# B&R Automation Studio project Parker_BMM_ST_V5_3147_V12 (part 28)

#### extruder.c - Implementation code
```c
/********************************************************************
 * COPYRIGHT --
 ********************************************************************
 * Program: extruder
 * File: extruder.c
 * Author: lij
 * Created: January 05, 2015
 ********************************************************************
 * Implementation of program extruder
 ********************************************************************/

#include <bur/plctypes.h>

#ifdef _DEFAULT_INCLUDES
#include <AsDefault.h>
#endif

/**************************************************************************************
** 					               include user files								 **
**************************************************************************************/
#include "edge.h"               /*edge function                         */
#include "keyap2100.h"
#include "pic_id.h"

/**************************************************************************************
** 					 	                 define								                   **
**************************************************************************************/
#define     S$EXTRUDER_WAIT		           	 0
#define     S$EXTRUDER_CONTACTOR_ON		   	10
#define     S$EXTRUDER_POWER_ON_DELAY			20
#define     S$EXTRUDER_POWER_ON		        	30
#define     S$EXTRUDER_READY		       		100
#define     S$EXTRUDER_BASIC_ZONE		  		110
#define     S$EXTRUDER_PRODUCTION_ZONE	   	130
#define     S$EXTRUDER_DEC_ZONE		       	150
#define     S$EXTRUDER_POWER_OFF_DECEL			200
#define     S$EXTRUDER_POWER_OFF_PROTECT		210
#define     S$EXTRUDER_POWER_OFF_DELAY			220
/**************************************************************************************
                               Function Declarations
**************************************************************************************/

/**************************************************************************************
     	        	       I N I T U P  O F   T H E   T A S K
**************************************************************************************/
void _INIT extruderINIT(void)
{
	/* TODO: Add code here */
	RTInfo_Task.enable = 1;
	RTInfo(&RTInfo_Task);

	tTask = RTInfo_Task.cycle_time/1000.0/1000.0;		/*  from us ---> s  */

	MotorSpeedA.minVal  	  = 0;
	MotorSpeedA.frequence	  = 30;
	MotorSpeedA.waitTimeSlow = 200;
	MotorSpeedA.waitTimeFast = 500;
	MotorSpeedA.unitsSlow    = 1;
	MotorSpeedA.unitsFast	= 5;
	MotorSpeedA.unitsVFast	= 20;

	MotorSpeedA.maxVal = 100;
	MotorSpeedA.minVal = 0;

	MotorSpeedB.minVal  	 = 0;
	MotorSpeedB.frequence	 = 30;
	MotorSpeedB.waitTimeSlow = 200;
	MotorSpeedB.waitTimeFast = 500;
	MotorSpeedB.unitsSlow    = 1;
	MotorSpeedB.unitsFast	 = 5;
	MotorSpeedB.unitsVFast	 = 20;

	MotorSpeedB.maxVal = 100;
	MotorSpeedB.minVal = 0;

	MotorSpeedVisu.frequence	= 30;
	MotorSpeedVisu.waitTimeSlow = 200;
	MotorSpeedVisu.waitTimeFast = 500;
	MotorSpeedVisu.unitsSlow    = 1;
	MotorSpeedVisu.unitsFast	= 5;
	MotorSpeedVisu.unitsVFast	= 20;

	MotorSpeedVisu.maxVal = 100;
	MotorSpeedVisu.minVal = 0;

	cntExtruderStopDelay = 0;

	gExtruderA.tTask  = tTask;
	gExtruderB.tTask  = tTask;
	gExtruderVisu.tTask = tTask;

	bHideCurrency = 1;
	bHideMeltTemp = 1;

	gExtruderA.Status.OnProtected = 1;
	gExtruderB.Status.OnProtected = 1;
	gExtruderC.Status.OnProtected = 1;
	gExtruderD.Status.OnProtected = 1;
	gExtruderVisu.Status.OnProtected = 1;

}
/**************************************************************************************
        				   C Y C L I C   P A R T   O F   T H E   T A S K
**************************************************************************************/
void _CYCLIC extruderCYCLIC(void)
{
	if(0 == gMachineFix.ExtruderA.RPM10v )gMachineFix.ExtruderA.RPM10v = 1500;
	if(0 == gMachineFix.ExtruderB.RPM10v )gMachineFix.ExtruderB.RPM10v  = 1500;
	if(0 == gMachineFix.ExtruderC.RPM10v )gMachineFix.ExtruderC.RPM10v = 1500;
	if(0 == gMachineFix.ExtruderD.RPM10v )gMachineFix.ExtruderD.RPM10v = 1500;
	if(0 == gMachineFix.ExtruderVisu.RPM10v )gMachineFix.ExtruderVisu.RPM10v = 1500;

	if(0 == gMachineFix.ExtruderA.Currency10V )gMachineFix.ExtruderA.Currency10V = 50;
	if(0 == gMachineFix.ExtruderB.Currency10V )gMachineFix.ExtruderB.Currency10V= 50;
	if(0 == gMachineFix.ExtruderC.Currency10V )gMachineFix.ExtruderC.Currency10V= 50;
	if(0 == gMachineFix.ExtruderD.Currency10V )gMachineFix.ExtruderD.Currency10V= 50;
	if(0 == gMachineFix.ExtruderVisu.Currency10V )gMachineFix.ExtruderVisu.Currency10V = 50;

	if((1 == gMachineFix.ExtruderD.Use) && 1 == gMachineFix.ExtruderVisu.Use)
	{

	}

	if(1 == gMachineFix.ExtruderD.Use && 1 == gMachineFix.ExtruderVisu.Use)
	{
		gMachineFix.ExtruderD.LinkWithMode = 1;
	}
	else
	{
		gMachineFix.ExtruderD.LinkWithMode = 0;
	}
	gMachineFix.ExtruderVisu.LinkWithMode = gMachineFix.ExtruderD.LinkWithMode;

	/*------------- CtrlType--------------- */
	gMachineFix.ExtruderB.eCtrlType = gMachineFix.ExtruderA.eCtrlType;
	gMachineFix.ExtruderC.eCtrlType = gMachineFix.ExtruderA.eCtrlType;
	gMachineFix.ExtruderD.eCtrlType = gMachineFix.ExtruderA.eCtrlType;
	gMachineFix.ExtruderVisu.eCtrlType = gMachineFix.ExtruderA.eCtrlType;

	if(1 == gEnableAll_HMI)
	{
		gEnableAll_HMI = 0;
		if(1 == gMachineFix.ExtruderA.Use) 		gExtruderHMI_Enable[0]=1;
		if(1 == gMachineFix.ExtruderB.Use) 		gExtruderHMI_Enable[1]=1;
		if(1 == gMachineFix.ExtruderC.Use) 		gExtruderHMI_Enable[2]=1;
		if(1 == gMachineFix.ExtruderD.Use) 		gExtruderHMI_Enable[3]=1;
		if(1 == gMachineFix.ExtruderVisu.Use) 	gExtruderHMI_Enable[4]=1;
	}
	else if( 1 == gDisableAll_HMI || 1 == gMachineIn.ExtruderNormal ||
		1 == gMachineIn.ExtrA_MotorErr || 1 == gMachineIn.ExtrB_MotorErr || 1 == gMachineIn.ExtrC_MotorErr ||
		1 == gMachineIn.ExtrD_MotorErr || 1 == gMachineIn.ExtrV_MotorErr)
	{
		gDisableAll_HMI = 0;
		if ( 1 == gMachineIn.ExtruderNormal)	gAlarm.ExtruderNormal = 1;
		gExtruderHMI_Enable[0] = 0;
		gExtruderHMI_Enable[1] = 0;
		gExtruderHMI_Enable[2] = 0;
		gExtruderHMI_Enable[3] = 0;
		gExtruderHMI_Enable[4] = 0;
	}

	/*  -------------------- Extruder motor speed and current -------------------------- */
	if(CTRL_VF == gMachineFix.ExtruderA.eCtrlType )// Analog VF Control
	{
		/*-------- Extruder A Use-------*/
		if(1 == gMachineFix.ExtruderA.Use)
		{
			// SetSpd condition
			if (1 == gExtruderHMI_Enable[0] && 1 == gMachineOut.ExtrA_On)
			{
				gExtruderA.aoSetRPM = (gMachinePara.ExtruderA.SetSpeed / gMachineFix.ExtruderA.RPM10v)*32767.0;
			}
			else
			{
				gExtruderA.aoSetRPM = 0;
			}

			// motor speed
			gExtruderA.ActRPM  = gExtruderA.aiActRPM/32767.0  * gMachineFix.ExtruderA.RPM10v;
			gExtruderA.Current = gExtruderA.aiCurrent/32767.0 * gMachineFix.ExtruderA.Currency10V;

			//Screw speed
			if (0 == gMachineFix.ExtruderA.Ratio)
			{
				gMachineFix.ExtruderA.Ratio =1;
			}
			else
			{
				gExtruderA.ActSpeed = gExtruderA.ActRPM /gMachineFix.ExtruderA.Ratio;
			}
		}
		else
		{
			gExtruderA.ActRPM = 0.0;
			gExtruderA.Current = 0.0;
		}

		/*-------- Extruder B Use-------*/
		if(1 == gMachineFix.ExtruderB.Use)
		{
			// SetSpd condition
			if (1 == gExtruderHMI_Enable[1] && 1 == gMachineOut.ExtrB_On)
			{
				gExtruderB.aoSetRPM = (gMachinePara.ExtruderB.SetSpeed / gMachineFix.ExtruderB.RPM10v)*32767.0;
			}
			else
			{
				gExtruderB.aoSetRPM = 0;
			}

			// motor speed
			gExtruderB.ActRPM = gExtruderB.aiActRPM/32767.0  * gMachineFix.ExtruderB.RPM10v;
			gExtruderB.Current = gExtruderB.aiCurrent/32767.0 * gMachineFix.ExtruderB.Currency10V;

			//Screw speed
			if (0 == gMachineFix.ExtruderB.Ratio)
			{
				gMachineFix.ExtruderB.Ratio =1;
			}
			else
			{
				gExtruderB.ActSpeed = gExtruderB.ActRPM /gMachineFix.ExtruderB.Ratio;
			}
		}
		else
		{
			gExtruderB.ActRPM = 0.0;
			gExtruderB.Current = 0.0;
		}

		/*-------- Extruder C Use-------*/
		if(1 == gMachineFix.ExtruderC.Use)
		{
			// SetSpd condition
			if (1 == gExtruderHMI_Enable[2] && 1 == gMachineOut.ExtrC_On)
			{
				gExtruderC.aoSetRPM = (gMachinePara.ExtruderC.SetSpeed / gMachineFix.ExtruderC.RPM10v)*32767.0;
			}
			else
			{
				gExtruderC.aoSetRPM = 0;
			}

			// motor speed
			gExtruderC.ActRPM = gExtruderC.aiActRPM/32767.0  * gMachineFix.ExtruderC.RPM10v;
			gExtruderC.Current = gExtruderC.aiCurrent/32767.0 * gMachineFix.ExtruderC.Currency10V;

			//Screw speed
			if (0 == gMachineFix.ExtruderC.Ratio)
			{
				gMachineFix.ExtruderC.Ratio =1;
			}
			else
			{
				gExtruderC.ActSpeed = gExtruderC.ActRPM /gMachineFix.ExtruderC.Ratio;
			}
		}
		else
		{
			gExtruderC.ActRPM = 0.0;
			gExtruderC.Current = 0.0;
		}

		/*-------- Extruder D Use-------*/
		if(1 == gMachineFix.ExtruderD.Use)
		{
			// SetSpd condition
			if (1 == gExtruderHMI_Enable[3] && 1 == gMachineOut.ExtrD_On)
			{
				gExtruderD.aoSetRPM = (gMachinePara.ExtruderD.SetSpeed / gMachineFix.ExtruderD.RPM10v)*32767.0;
			}
			else
			{
				gExtruderD.aoSetRPM = 0;
			}

			// motor speed
			gExtruderD.ActRPM = gExtruderD.aiActRPM/32767.0  * gMachineFix.ExtruderD.RPM10v;
			gExtruderD.Current = gExtruderD.aiCurrent/32767.0 * gMachineFix.ExtruderD.Currency10V;

			//Screw speed
			if (0 == gMachineFix.ExtruderD.Ratio)
			{
				gMachineFix.ExtruderD.Ratio =1;
			}
			else
			{
				gExtruderD.ActSpeed = gExtruderD.ActRPM /gMachineFix.ExtruderD.Ratio;
			}
		}
		else
		{
			gExtruderD.ActRPM = 0.0;
			gExtruderD.Current = 0.0;
		}

		/*-------- Extruder Visu Use-------*/
		if(1 == gMachineFix.ExtruderVisu.Use)
		{
			// SetSpd condition
			if (1 == gExtruderHMI_Enable[4] && 1 == gMachineOut.ExtrVisu_On)
			{
				gExtruderVisu.aoSetRPM = (gMachinePara.ExtruderVisu.SetSpeed / gMachineFix.ExtruderVisu.RPM10v)*32767.0;
			}
			else
			{
				gExtruderVisu.aoSetRPM = 0;
			}

			// motor speed
			gExtruderVisu.ActRPM = gExtruderVisu.aiActRPM/32767.0  * gMachineFix.ExtruderVisu.RPM10v;
			gExtruderVisu.Current = gExtruderVisu.aiCurrent/32767.0 * gMachineFix.ExtruderVisu.Currency10V;

			//Screw speed
			if (0 == gMachineFix.ExtruderVisu.Ratio)
			{
				gMachineFix.ExtruderVisu.Ratio =1;
			}
			else
			{
				gExtruderVisu.ActSpeed = gExtruderVisu.ActRPM /gMachineFix.ExtruderVisu.Ratio;
			}
		}
		else
		{
			gExtruderVisu.ActRPM = 0.0;
			gExtruderVisu.Current = 0.0;
		}

	}

	/* ------------------------ Extruder Protect Delay Switch On  ---------------------------- */
	/* ----- A extruder ----- */
	if(0 == gExtruderA.Status.OnProtected  && 0 == gMachineOut.ExtrA_On )
	{
		gMacTimer.ExtrA_OnDelay.IN = 1;
		gMacTimer.ExtrA_OnDelay.PT = gMachineFix.ExtruderA.tProtect*100;

		if(1 == gMacTimer.ExtrA_OnDelay.Q)
		{
			gMacTimer.ExtrA_OnDelay.IN = 0;
			gExtruderA.Status.OnProtected = 1;
		}
	}
	else if( 1 == gMachineOut.ExtrA_On )
	{
		gExtruderA.Status.OnProtected = 0;
	}

	/* ----- B extruder ----- */
	if(0 == gExtruderB.Status.OnProtected  && 0 == gMachineOut.ExtrB_On )
	{
		gMacTimer.ExtrB_OnDelay.IN = 1;
		gMacTimer.ExtrB_OnDelay.PT = gMachineFix.ExtruderB.tProtect*100;

		if(1 == gMacTimer.ExtrB_OnDelay.Q)
		{
			gMacTimer.ExtrB_OnDelay.IN = 0;
			gExtruderB.Status.OnProtected = 1;
		}
	}
	else if( 1 == gMachineOut.ExtrB_On )
	{
		gExtruderB.Status.OnProtected = 0;
	}

	/* ----- C extruder ----- */
	if(0 == gExtruderC.Status.OnProtected && 0 == gMachineOut.ExtrC_On )
	{
		gMacTimer.ExtrC_OnDelay.IN = 1;
		gMacTimer.ExtrC_OnDelay.PT = gMachineFix.ExtruderC.tProtect*100;

		if(1 == gMacTimer.ExtrC_OnDelay.Q)
		{
			gMacTimer.ExtrC_OnDelay.IN = 0;
			gExtruderC.Status.OnProtected = 1;
		}
	}
	else if( 1 == gMachineOut.ExtrC_On )
	{
		gExtruderC.Status.OnProtected = 0;
	}

	/* ----- D extruder ----- */
	if(0 == gExtruderD.Status.OnProtected && 0 == gMachineOut.ExtrD_On )
	{
		gMacTimer.ExtrD_OnDelay.IN = 1;
		gMacTimer.ExtrD_OnDelay.PT = gMachineFix.ExtruderD.tProtect*100;

		if(1 == gMacTimer.ExtrD_OnDelay.Q)
		{
			gMacTimer.ExtrD_OnDelay.IN = 0;
			gExtruderD.Status.OnProtected = 1;
		}
	}
	else if( 1 == gMachineOut.ExtrD_On )
	{
		gExtruderD.Status.OnProtected = 0;
	}

	/* ----- V extruder ----- */
	if(0 == gExtruderVisu.Status.OnProtected && 0 == gMachineOut.ExtrVisu_On )
	{
		gMacTimer.ExtrVisu_OnDelay.IN = 1;
		gMacTimer.ExtrVisu_OnDelay.PT = gMachineFix.ExtruderVisu.tProtect*100;

		if(1 == gMacTimer.ExtrVisu_OnDelay.Q)
		{
			gMacTimer.ExtrVisu_OnDelay.IN = 0;
			gExtruderVisu.Status.OnProtected = 1;
		}
	}
	else if( 1 == gMachineOut.ExtrVisu_On )
	{
		gExtruderVisu.Status.OnProtected = 0;
	}

	/* ----------------------- Switch On extruder ----------------------- */
	if(gPanelObj.GetPicture != PIC_INIT && gPanelObj.GetPicture != PIC_SCREEN_SAVE)
	{
		/*	-----------Extruder A ----------*/
		if(1 == EDGEPOS(gPanelObj.KeyMatric[S$KEYMATRIX_EXTRUDER_A_ABB],PKeyMatric[S$KEYMATRIX_EXTRUDER_A_ABB]))
			{
			if (1==gMachineFix.ExtruderA.Use)
			{
				if (0==gExtruderTempLow_HMIFlag && 0 == gMachineInfo.DieLipTempLow)  //ipis0718
				{
					if (0==gMachineInfo.bLoweringFlag)  //ipis0614
					{
						if(1 == gExtruderA.Status.OnProtected || 1 == gMachineOut.ExtrA_On)
						{
							gMachineOut.ExtrA_On = !gMachineOut.ExtrA_On; //DO
						}
						else
						{
							gImply.ExtrA_OnDelay = 1;
						}
					}
					else
					{
						gImply.TempLoweringEnable =1;
					}
				}
				else
				{
					gImply.TempLow = gExtruderTempLow_HMIFlag;
					gImply.DieLipTempLow = gMachineInfo.DieLipTempLow;
				}
			}
			else
			{
				gMachineOut.ExtrA_On =0;
				gImply.ExtruderNoChoose =1;
			}
		}

		/*	-----------Extruder B ----------*/
		if(1 == EDGEPOS(gPanelObj.KeyMatric[S$KEYMATRIX_EXTRUDER_B_ABB],PKeyMatric[S$KEYMATRIX_EXTRUDER_B_ABB]))
			{
			if (1==gMachineFix.ExtruderB.Use)
			{
				if (0==gExtruderTempLow_HMIFlag && 0 == gMachineInfo.DieLipTempLow)  //ipis0718
				{
					if (0==gMachineInfo.bLoweringFlag) //ipis0614
					{
						if(1 == gExtruderB.Status.OnProtected || 1 == gMachineOut.ExtrB_On) //owen 20200921
						{
							gMachineOut.ExtrB_On = !gMachineOut.ExtrB_On; //DO
						}
						else
						{
							gImply.ExtrB_OnDelay = 1;
						}
					}
					else
					{
						gImply.TempLoweringEnable =1;
					}
				}
				else
				{
					gImply.TempLow = gExtruderTempLow_HMIFlag;
					gImply.DieLipTempLow = gMachineInfo.DieLipTempLow;
				}
			}
			else
			{
				gMachineOut.ExtrB_On=0;
				gImply.ExtruderNoChoose =1;
			}
		}

		/*	-----------Extruder C ----------*/
		if(1 == EDGEPOS(gPanelObj.KeyMatric[S$KEYMATRIX_EXTRUDER_C_ABB],PKeyMatric[S$KEYMATRIX_EXTRUDER_C_ABB]))
			{

			if (1==gMachineFix.ExtruderC.Use)
			{
				if (0==gExtruderTempLow_HMIFlag && 0 == gMachineInfo.DieLipTempLow)  //ipis0718
				{
					if (0==gMachineInfo.bLoweringFlag) //ipis0614
					{
						if(1 == gExtruderC.Status.OnProtected || 1 == gMachineOut.ExtrC_On) //owen 20200921
						{
							gMachineOut.ExtrC_On =!gMachineOut.ExtrC_On; //DO
						}
						else
						{
							gImply.ExtrC_OnDelay = 1;
						}
					}
					else
					{
						gImply.TempLoweringEnable =1;
					}
				}
				else
				{
					gImply.TempLow = gExtruderTempLow_HMIFlag;
					gImply.DieLipTempLow = gMachineInfo.DieLipTempLow;
				}
			}
			else
			{
				gMachineOut.ExtrC_On =0;
				gImply.ExtruderNoChoose =1;
			}
		}

		/*	-----------Extruder D ----------*/
		if(1 == EDGEPOS(gPanelObj.KeyMatric[S$KEYMATRIX_EXTRUDER_D_ABB],PKeyMatric[S$KEYMATRIX_EXTRUDER_D_ABB]))
			{
			if (1==gMachineFix.ExtruderD.Use)
			{
				if (0==gExtruderTempLow_HMIFlag && 0 == gMachineInfo.DieLipTempLow)  //ipis0718
				{
					if (0==gMachineInfo.bLoweringFlag) //ipis0614
					{

						if(1 == gExtruderD.Status.OnProtected || 1 == gMachineOut.ExtrD_On) //owen 20200921
						{
							gMachineOut.ExtrD_On =!gMachineOut.ExtrD_On; //DO
						}
						else
						{
							gImply.ExtrD_OnDelay = 1;
						}
					}
					else
					{
						gImply.TempLoweringEnable =1;
					}

				}
				else
				{
					gImply.TempLow = gExtruderTempLow_HMIFlag;
					gImply.DieLipTempLow = gMachineInfo.DieLipTempLow;
				}
			}
			else
			{
				gMachineOut.ExtrD_On =0;
				gImply.ExtruderNoChoose =1;
			}

		}

		/*	-----------Extruder Visu ----------*/
		if (1 == gMachineFix.ExtruderD.LinkWithMode)
		{
			if(1 == EDGEPOS(gPanelObj.KeyMatric[S$KEYMATRIX_EXTRUDER_D_ABB],PKeyMatric[S$KEYMATRIX_EXTRUDER_V_ABB]))
				{
				if (1==gMachineFix.ExtruderVisu.Use)
				{
					if (0==gExtruderTempLow_HMIFlag && 0 == gMachineInfo.DieLipTempLow)  //ipis0718
					{
						if (0==gMachineInfo.bLoweringFlag) //ipis0614
						{
							if(1 == gExtruderD.Status.OnProtected )  //from  extruder D switch on delay
							{
								if(1 == gExtruderVisu.Status.OnProtected || 1 == gMachineOut.ExtrVisu_On) //owen 20200921
								{
									gMachineOut.ExtrVisu_On =!gMachineOut.ExtrVisu_On; //DO
								}
								else
								{
									gImply.ExtrVisu_OnDelay = 1;
								}
							}
							else
							{
								gImply.ExtrD_OnDelay = 1;
							}
						}
						else
						{
							gImply.TempLoweringEnable =1;
						}
					}
					else
					{
						gImply.TempLow = gExtruderTempLow_HMIFlag;
						gImply.DieLipTempLow = gMachineInfo.DieLipTempLow;
					}
				}
				else
				{
					gMachineOut.ExtrVisu_On=0;
					gImply.ExtruderNoChoose =1;
				}
			}

		}
		else
		{
			if(1 == EDGEPOS(gPanelObj.KeyMatric[S$KEYMATRIX_EXTRUDER_V_ABB],PKeyMatric[S$KEYMATRIX_EXTRUDER_V_ABB]))
				{
				if (1==gMachineFix.ExtruderVisu.Use)
				{
					if (0==gExtruderTempLow_HMIFlag && 0 == gMachineInfo.DieLipTempLow)  //ipis0718
					{
						if (0==gMachineInfo.bLoweringFlag) //ipis0614
						{
							if(1 == gExtruderVisu.Status.OnProtected || 1 == gMachineOut.ExtrVisu_On) //owen 20200921
							{
								gMachineOut.ExtrVisu_On =!gMachineOut.ExtrVisu_On; //DO
							}
							else
							{
								gImply.ExtrVisu_OnDelay = 1;
							}
						}
						else
						{
							gImply.TempLoweringEnable =1;
						}
					}
					else
					{
						gImply.TempLow = gExtruderTempLow_HMIFlag;
						gImply.DieLipTempLow = gMachineInfo.DieLipTempLow;
					}
				}
				else
				{
					gMachineOut.ExtrVisu_On=0;
					gImply.ExtruderNoChoose =1;
				}
			}
		}

	}

	/*	----------------------------------------------------------------------------------------------------------------------*/

	gMachineInfo.Extruder       = gMachineOut.ExtrA_On;
	gMachineOut.ExtruderCooling = gMachineInfo.Extruder;

	/*	-------------------------------------------------------------- */
	/*  ---------------------- Stop extruder ------------------------- */
	/*	-------------------------------------------------------------- */
	/* ----- A extruder ----- */
	gExtruderA.bKeyOff = 0;
	if (1 == gMachineInfo.ExtrTLow     || 0 == gMachineInfo.IsHeat        	 || 1 == gMachineInfo.DieLipTempLow   /*|| 0 == gMachineIn.ParisonPumpRunning*/
		|| 1 == gMachineIn.ExtrA_MotorErr || 0 == gMachineIn.ExtrA_Wire_MotorErr || 1 == gMachineIn.ExtrA_CoolMotorErr || 1 == gMachineIn.InstancyStop || 1 == gMachineInfo.SafeInStop)
		/*|| 1 == gAlarm.A_ColiTempNormal   ||1 == gAlarm.A_ExtrMotorTempStop     || 1 == gAlarm.ExtrAMeltP */ // 2018.06.05 Jack: Add ExtrAMeltP alarm stop condition
	{
		if(1 == gMachineOut.ExtrA_On)
		{
			if(1 == gMachineInfo.ExtrTLow)gAlarm.ScrewTempLow = 1;
			if(0 == gMachineInfo.IsHeat)gAlarm.HeatingNotOn = 1;
			gAlarm.DieLipTempLow = gMachineInfo.DieLipTempLow;
			//		if(0 == gMachineIn.ParisonPumpRunning)gAlarm.ParisonPumpNotOn = 1;
			if ( 1 == gMachineIn.ExtrA_MotorErr ||0 == gMachineIn.ExtrA_Wire_MotorErr)	gAlarm.A_ExtruderMotorOverload =1;  //ipis0323

			//		gAlarm.A_ExtruderMotorOverload = gMachineIn.ExtrA_MotorErr;
			gExtruderA.bKeyOff = 1;
			gMachineOut.ExtrA_On =0;
			gMachineInfo.ExtrA_ErrStop_LinkWith = 1;  //Extruder Link With Selection
		}
	}

	/* ----- B extruder ----- */
	gExtruderB.bKeyOff = 0;
	if (1 == gMachineInfo.ExtrTLow     || 0 == gMachineInfo.IsHeat        	 || 1 == gMachineInfo.DieLipTempLow   /*|| 0 == gMachineIn.ParisonPumpRunning*/
	 || 1 == gMachineIn.ExtrB_MotorErr || 0 == gMachineIn.ExtrB_Wire_MotorErr || 1 == gMachineIn.ExtrB_CoolMotorErr ||1==gMachineIn.InstancyStop || 1 == gMachineInfo.SafeInStop)
	{
		if(1 == gMachineOut.ExtrB_On)
		{
			if(1 == gMachineInfo.ExtrTLow)gAlarm.ScrewTempLow = 1;
			if(0 == gMachineInfo.IsHeat)gAlarm.HeatingNotOn = 1;
			gAlarm.DieLipTempLow = gMachineInfo.DieLipTempLow;
			//	if(0 == gMachineIn.ParisonPumpRunning)gAlarm.ParisonPumpNotOn = 1;
			if (  1 == gMachineIn.ExtrB_MotorErr ||0 == gMachineIn.ExtrB_Wire_MotorErr)	gAlarm.B_ExtruderMotorOverload =1;  //ipis0323

			//		gAlarm.B_ExtruderMotorOverload = gMachineIn.ExtrB_MotorErr;
			gExtruderB.bKeyOff = 1;
			gMachineOut.ExtrB_On =0;
		}
	}

	/* ----- C extruder ----- */
	gExtruderC.bKeyOff = 0;
	if (1 == gMachineInfo.ExtrTLow     || 0 == gMachineInfo.IsHeat        	 || 1 == gMachineInfo.DieLipTempLow   /*|| 0 == gMachineIn.ParisonPumpRunning*/   ||
		1 == gMachineIn.ExtrC_MotorErr || 0 == gMachineIn.ExtrC_Wire_MotorErr || 1 == gMachineIn.ExtrC_CoolMotorErr ||1==gMachineIn.InstancyStop || 1 == gMachineInfo.SafeInStop )
	{
		if(1 == gMachineOut.ExtrC_On)
		{
			if(1 == gMachineInfo.ExtrTLow)gAlarm.ScrewTempLow = 1;
			if(0 == gMachineInfo.IsHeat)gAlarm.HeatingNotOn = 1;
			gAlarm.DieLipTempLow = gMachineInfo.DieLipTempLow;
			//	if(0 == gMachineIn.ParisonPumpRunning)gAlarm.ParisonPumpNotOn = 1;
			if (  1 == gMachineIn.ExtrC_MotorErr ||0 == gMachineIn.ExtrC_Wire_MotorErr)	gAlarm.C_ExtruderMotorOverload =1;  //ipis0323

			//			gAlarm.C_ExtruderMotorOverload = gMachineIn.ExtrC_MotorErr;

			gExtruderC.bKeyOff = 1;
			gMachineOut.ExtrC_On =0;
		}
	}

	/* ----- D extruder ----- */
	gExtruderD.bKeyOff = 0;
	if (1 == gMachineInfo.ExtrTLow     || 0 == gMachineInfo.IsHeat        	 || 1 == gMachineInfo.DieLipTempLow   /*|| 0 == gMachineIn.ParisonPumpRunning*/   ||
		1 == gMachineIn.ExtrD_MotorErr || 0 == gMachineIn.ExtrD_Wire_MotorErr|| 1 == gMachineIn.ExtrD_CoolMotorErr||1==gMachineIn.InstancyStop || 1 == gMachineInfo.SafeInStop)
	{
		if(1 == gMachineOut.ExtrD_On)
		{
			if(1 == gMachineInfo.ExtrTLow)gAlarm.ScrewTempLow = 1;
			if(0 == gMachineInfo.IsHeat)gAlarm.HeatingNotOn = 1;
			gAlarm.DieLipTempLow = gMachineInfo.DieLipTempLow;
			//			if(0 == gMachineIn.ParisonPumpRunning)gAlarm.ParisonPumpNotOn = 1;
			if (  1 == gMachineIn.ExtrD_MotorErr ||0 == gMachineIn.ExtrD_Wire_MotorErr)	gAlarm.D_ExtruderMotorOverload = 1;  //ipis0323

			//		gAlarm.B_ExtruderMotorOverload = gMachineIn.ExtrD_MotorErr;
			gExtruderD.bKeyOff = 1;
			gMachineOut.ExtrD_On =0;
			gMachineInfo.ExtrD_ErrStop_LinkWith = 1;   //Extruder Link With Selection
		}
	}

	/* ----- Visual extruder ----- */
	gExtruderVisu.bKeyOff = 0;
	if (1 == gMachineInfo.ExtrTLow     || 0 == gMachineInfo.IsHeat        	 || 1 == gMachineInfo.DieLipTempLow   /*|| 0 == gMachineIn.ParisonPumpRunning*/   ||
		1 == gMachineIn.ExtrV_MotorErr || 0 == gMachineIn.ExtrV_Wire_MotorErr|| 1 == gMachineIn.ExtrV_CoolMotorErr /*|| 0 == gMachineOut.ExtrA_On*/ ||1==gMachineIn.InstancyStop || 1 == gMachineInfo.SafeInStop)
	{
		if(1 == gMachineOut.ExtrVisu_On)
		{
			if(1 == gMachineInfo.ExtrTLow)gAlarm.ScrewTempLow = 1;
			if(0 == gMachineInfo.IsHeat)gAlarm.HeatingNotOn = 1;
			gAlarm.DieLipTempLow = gMachineInfo.DieLipTempLow;
			//	if(0 == gMachineIn.ParisonPumpRunning)gAlarm.ParisonPumpNotOn = 1;
			if (  1 == gMachineIn.ExtrV_MotorErr ||0 == gMachineIn.ExtrV_Wire_MotorErr)	gAlarm.VisuExtrMotorOverload =1;  //ipis0323

			//	gAlarm.VisuExtrMotorOverload = gMachineIn.ExtrV_MotorErr;
			gExtruderVisu.bKeyOff = 1;
			gMachineOut.ExtrVisu_On =0;
			gMachineInfo.ExtrVisu_ErrStop_LinkWith = 1;  //Extruder Link With Selection
		}
	}

	/* ----- All extruder ----- */

	/*	-------------------------------------------------------------- */
	/* ---------------- Extruder Link With Selection  ---------------- */
	/*	-------------------------------------------------------------- */
	/* ----- A extruder ----- */
	if(1 == gMachineFix.ExtruderA.LinkWithMode)
	{
		if( EDGENEG(gMachineOut.ExtrA_On,oldExtrA_On))
		{
			gMachineOut.ParisonPump = 0;
		}
		else if (1 == gMachineInfo.ExtrA_ErrStop_LinkWith)
		{
			gMachineInfo.ExtrA_ErrStop_LinkWith =0;
			gMachineOut.ParisonPump = 0;
		}
	}

	/* ----- D extruder ----- */
	if(1 == gMachineFix.ExtruderD.LinkWithMode)
	{
		if( EDGENEG(gMachineOut.ExtrD_On,oldExtrD_On))
		{
			gMachineOut.ExtrVisu_On = 0;
		}
		else if (1 == gMachineInfo.ExtrD_ErrStop_LinkWith)
		{
			gMachineInfo.ExtrD_ErrStop_LinkWith = 0;
			gMachineOut.ExtrVisu_On = 0;
		}
	}

	/* ----- Visu extruder ----- */
	if(1 == gMachineFix.ExtruderVisu.LinkWithMode)
	{
		if( EDGENEG(gMachineOut.ExtrVisu_On,oldExtrVisu_On))
		{
			gMachineOut.ExtrD_On = 0;
		}
		else if (1 == gMachineInfo.ExtrVisu_ErrStop_LinkWith)
		{
			gMachineInfo.ExtrVisu_ErrStop_LinkWith =0;
			gMachineOut.ExtrD_On = 0;
		}
	}

	oldExtrA_On = gMachineOut.ExtrA_On;
	oldExtrB_On = gMachineOut.ExtrB_On;
	oldExtrC_On = gMachineOut.ExtrC_On;
	oldExtrD_On = gMachineOut.ExtrD_On;
	oldExtrVisu_On = gMachineOut.ExtrVisu_On;

	/* ------------------------ Auto error stop extruder ---------------------------- */
	if(1 == gPROCESS_info.extruderStopEnable)
	{
		cntExtruderStopDelay ++;
	}
	else
	{
		cntExtruderStopDelay = 0;
	}

	if(gMachineFix.ExtruderA.StopTime <= 0.0)gMachineFix.ExtruderA.StopTime = 3.0;
	if(gMachineFix.ExtruderA.StopTime < cntExtruderStopDelay * tTask)
	{
		if(1 == gTKmanual.Status)
		{
			gDisableAll_HMI 				=1;	  //ipis0719
			//			gMachineOut.ExtrA_On =0;
			//			gMachineOut.ExtrB_On =0;
			//			gMachineOut.ExtrD_On =0;
			//			gMachineOut.ExtrVisu_On =0;
			gExtruderA.bKeyOff = 1;
			gExtruderB.bKeyOff = 1;
			gExtruderC.bKeyOff = 1;
			gExtruderD.bKeyOff =1;
			gExtruderVisu.bKeyOff = 1;
			gPROCESS_info.extruderStopEnable = 0;
			cntExtruderStopDelay = 0;
		}
	}
}
/**************************************************************************************
        				   E X I T   P A R T   O F   T H E   T A S K
**************************************************************************************/
void _EXIT extruderEXIT(void)
{
	/* TODO: Add code here */
}
```

#### extruder.var - Local variables
```iecst
(********************************************************************
 * COPYRIGHT --
 ********************************************************************
 * Program: extruder
 * File: extruder.var
 * Author: lij
 * Created: January 05, 2015
 ********************************************************************
 * Local variables of program extruder
 ********************************************************************)
VAR
	tTask : REAL := 0.0;
	RTInfo_Task : RTInfo := (0);
	tAlarmExtrTempA : REAL;
	tStopExtrTempA : REAL;
	tColiTempNormalA : REAL;
	bHideCurrency : UINT;
	bHideMeltTemp : UINT;
	btnZeroExtrA : USINT;
	btnMaxExtrA : USINT;
	tMaxExtrA : REAL;
	tZeroExtrA : REAL;
	btnZeroExtrB : USINT;
	btnMaxExtrB : USINT;
	tMaxExtrB : REAL;
	ExtrA_HopperKeyOld : USINT;
	ExtrB_HopperKeyOld : USINT;
	LubricCheckA : Lubricate_Check_typ;
	LubricCheckB : Lubricate_Check_typ;
	LubricCheckVisu : Lubricate_Check_typ;
	MotorSpeedA : speedAdjust_typ;
	MotorSpeedB : speedAdjust_typ;
	MotorSpeedVisu : speedAdjust_typ;
	tExtrA_OnNormal : REAL;
	tExtrB_OnNormal : REAL;
	tExtrV_OnNormal : REAL;
	cntExtruderStopDelay : UDINT;
	PKeyMatric : ARRAY[0..MAX_KEY_COUNT] OF USINT;
	NKeyMatric : ARRAY[0..MAX_KEY_COUNT] OF USINT;
	oldExtrA_On : USINT;
	oldExtrB_On : USINT;
	oldExtrC_On : USINT;
	oldExtrD_On : USINT;
	oldExtrVisu_On : USINT;
END_VAR
```

- edge.h (reference to Logical/GlobalIncludes/edge.h)

### Program Logical/machine/clean (ANSIC, version 1.00.0) - clean proportional valve

#### clean.c
```c
/********************************************************************
 * COPYRIGHT --  B&R China
 ********************************************************************
 * Program: clean
 * File: clean.c
 * Author: lijianjun
 * Created: March 06, 2013
 ********************************************************************
 * Implementation of program clean --- clean proportional  valve
 ********************************************************************/

#include <bur/plctypes.h>

#ifdef _DEFAULT_INCLUDES
	#include <AsDefault.h>
#endif

#include "defines.h"
#include "edge.h"
#include "keyap2100.h"
//#include "keyap880.h"
#include "pic_id.h"

/**************************************************************************************
                            Function Declarations
**************************************************************************************/
void CleanValveCtrl (CleanValve_typ * pCleanValveFix,CleanCtrl_typ * pCtrl, timer_typ *tValveCleanTotal,timer_typ *tValveClean,UINT *pMold_Step);

/**************************************************************************************
     	        		         I N I T U P  O F   T H E   T A S K
**************************************************************************************/
void _INIT cleanvlave_init(void)
{
	RClampCleanValveCtrl.Step = 3000;
	RCarriageCleanValveCtrl.Step = 3000;
}  /* end of _INIT */
/**************************************************************************************
****				         C Y C L I C   P A R T   O F   T H E   T A S K
**************************************************************************************/
void _CYCLIC cleanvlave_cyclic(void)
{
	/*----------------------------------*/
	/*-------------Clamp----------------*/
	/*----------------------------------*/
	if(VALVE_PROP == gMachineFix.MoldR.Clamp.eValveType)
	{
		if(RClampCleanValveCtrl.Step >= 10 && RClampCleanValveCtrl.Step <= 3000)
		{
			//Valve Out
			RMold.ValveOut.ClampOpn 		= RClampCleanValveCtrl.ValveOut.ValveFw1;
			RMold.ValveOut.ClampOpnRelease 	= RClampCleanValveCtrl.ValveOut.ValveFw2;

			RMold.ValveOut.ClampCls 	= RClampCleanValveCtrl.ValveOut.ValveBw1;
			//Pressure
			RMold.Clamp.p_set = RClampCleanValveCtrl.p_set;
		}
		if(LClampCleanValveCtrl.Step >= 10 && LClampCleanValveCtrl.Step <= 3000)
		{
			//Valve Out
			LMold.ValveOut.ClampOpn 		= LClampCleanValveCtrl.ValveOut.ValveFw1;
			LMold.ValveOut.ClampOpnRelease 	= LClampCleanValveCtrl.ValveOut.ValveFw2;

			LMold.ValveOut.ClampCls 	= LClampCleanValveCtrl.ValveOut.ValveBw1;
			//Pressure
			LMold.Clamp.p_set = LClampCleanValveCtrl.p_set;
		}
		CleanValveCtrl(&gMachineFix.CleanValve.MoldR.Clamp,&RClampCleanValveCtrl,&gMacTimer.RClampValveCleanTotal,&gMacTimer.RClampValveClean,&RMold.Clamp.Step);
		CleanValveCtrl(&gMachineFix.CleanValve.MoldL.Clamp,&LClampCleanValveCtrl,&gMacTimer.LClampValveCleanTotal,&gMacTimer.LClampValveClean,&LMold.Clamp.Step);
	}

	/*----------------------------------*/
	/*-------------Carriage-------------*/
	/*----------------------------------*/
	if(VALVE_PROP == gMachineFix.MoldR.Carriage.eValveType)
	{
		if(RCarriageCleanValveCtrl.Step >= 10 && RCarriageCleanValveCtrl.Step <= 3000)
		{
			//Valve Out
			RMold.ValveOut.CarriageFw = RCarriageCleanValveCtrl.ValveOut.ValveFw1;
			RMold.ValveOut.CarriageBw = RCarriageCleanValveCtrl.ValveOut.ValveBw1;
			//Pressure
			RMold.Carriage.p_set = RCarriageCleanValveCtrl.p_set;
		}
		if(LCarriageCleanValveCtrl.Step >= 10 && LCarriageCleanValveCtrl.Step <= 3000)
		{
			//Valve Out
			LMold.ValveOut.CarriageFw = LCarriageCleanValveCtrl.ValveOut.ValveFw1;
			LMold.ValveOut.CarriageBw = LCarriageCleanValveCtrl.ValveOut.ValveBw1;
			//Pressure
			LMold.Carriage.p_set = LCarriageCleanValveCtrl.p_set;
		}
		CleanValveCtrl(&gMachineFix.CleanValve.MoldR.Carriage,&RCarriageCleanValveCtrl,&gMacTimer.RCarriageValveCleanTotal,&gMacTimer.RCarriageValveClean,&RMold.Carriage.Step);
		CleanValveCtrl(&gMachineFix.CleanValve.MoldL.Carriage,&LCarriageCleanValveCtrl,&gMacTimer.LCarriageValveCleanTotal,&gMacTimer.LCarriageValveClean,&LMold.Carriage.Step);
	}

	/*----------------------------------*/
	/*-------------Blowpin--------------*/
	/*----------------------------------*/
//	if(RBlowPinCleanValveCtrl.Step >= 10 && RBlowPinCleanValveCtrl.Step <= 3000)
//	{
//		//Valve Out
//		RMold.ValveOut.BlowPinDn = RBlowPinCleanValveCtrl.ValveOut.ValveFw1;
//		RMold.ValveOut.BlowPinUp = RBlowPinCleanValveCtrl.ValveOut.ValveBw1;
//		//Pressure
//		RMold.BlowPin.p_set = RBlowPinCleanValveCtrl.p_set;
//	}
//	if(LBlowPinCleanValveCtrl.Step >= 10 && LBlowPinCleanValveCtrl.Step <= 3000)
//	{
//		//Valve Out
//		LMold.ValveOut.BlowPinDn = LBlowPinCleanValveCtrl.ValveOut.ValveFw1;
//		LMold.ValveOut.BlowPinUp = LBlowPinCleanValveCtrl.ValveOut.ValveBw1;
//		//Pressure
//		LMold.BlowPin.p_set = LBlowPinCleanValveCtrl.p_set;
//	}
//	CleanValveCtrl(&gMachineFix.CleanValve.MoldR.BlowPin,&RBlowPinCleanValveCtrl,&gMacTimer.RBlowPinValveCleanTotal,&gMacTimer.RBlowPinValveClean,&RMold.BlowPin.Step);
//	CleanValveCtrl(&gMachineFix.CleanValve.MoldL.BlowPin,&LBlowPinCleanValveCtrl,&gMacTimer.LBlowPinValveCleanTotal,&gMacTimer.LBlowPinValveClean,&LMold.BlowPin.Step);

}  /* end of _CYCLIC */

void CleanValveCtrl(CleanValve_typ * pCleanValveFix,CleanCtrl_typ * pCtrl, timer_typ *tValveCleanTotal,timer_typ *tValveClean,UINT *pMold_Step)
{

		if( 1 == pCtrl->Enable && 0 == pCtrl->Enable)
		{
			if(PIC_OEM_SETTING_10 == gPanelObj.GetPicture)
			{
				pCtrl->Enable = 1;
			}
		}
		/* Start clean valve  */
		if(gPanelObj.PasswordLevel > 2 && 1 == gTKcalib.Status)
		{
			if(1 == pCtrl->Enable)
			{
				pCtrl->Enable = 0;

				if(pCtrl->Step != 0)
				{
					pCtrl->Step = 3000;
					*pMold_Step = 0;
				}
				else
				{
					pCtrl->Step = 10;
					*pMold_Step = 5;  /*Clean Valve Step*/
				}
			}
		}/* if(gPanelObj.PasswordLevel > 3) */

		pCtrl->oldEnable  =  pCtrl->Enable;

	/*  step machine clear valve */
	switch(pCtrl->Step)
	{
		case 0: 	// Off

			break;

		case 10: 	// total time start
			tValveCleanTotal->IN = 1;
			tValveCleanTotal->PT = pCleanValveFix->CleanValveTotalTime*60;
			pCtrl->Step = 100;
			break;

		case 100:	//Fw Timer Setting
			tValveClean->IN = 1;
			tValveClean->PT = pCleanValveFix->CleanValveFwTime;
			pCtrl->Step = 200;
			break;

		case 200:	//Fw
			pCtrl->ValveOut.ValveFw1 = 1;
			pCtrl->ValveOut.ValveFw2 = 1;

			pCtrl->p_set = pCtrl->Para.P_FwClean;
			pCtrl->TimeDis.CleanValveFwDis = tValveClean->ET;
			if(1 == tValveClean->Q)
			{
				pCtrl->TimeDis.CleanValveFwDis = 0;
				tValveClean->IN = 0;
				pCtrl->Step = 300;
			}
			break;

		case 300:	//Fw End
			pCtrl->ValveOut.ValveFw1 = 0;
			pCtrl->ValveOut.ValveFw2 = 0;

			pCtrl->p_set = 0;

			pCtrl->Step = 400;
			break;

		case 400:	//Interval Timer Setting
			tValveClean->IN = 1;
			tValveClean->PT = pCleanValveFix->CleanValveInterval;
			pCtrl->Step = 500;
			break;

		case 500:	//Interval
			pCtrl->TimeDis.CleanValveIntervalDis = tValveClean->ET;
			if(1 == tValveClean->Q)
			{
				pCtrl->TimeDis.CleanValveIntervalDis = 0;
				tValveClean->IN = 0;
				pCtrl->Step = 600;
			}

			break;

		case 600:
			pCtrl->Step = 700;
			break;

		case 700:	//Bw Timer Setting
			tValveClean->IN = 1;
			tValveClean->PT = pCleanValveFix->CleanValveBwTime;
			pCtrl->Step = 800;
			break;

		case 800:	//Bw
			pCtrl->ValveOut.ValveBw1 = 1;
			pCtrl->ValveOut.ValveBw2 = 1;

			pCtrl->p_set = pCtrl->Para.P_BwClean;
			pCtrl->TimeDis.CleanValveBwDis = tValveClean->ET;
			if(1 == tValveClean->Q)
			{
				pCtrl->TimeDis.CleanValveBwDis = 0;
				tValveClean->IN = 0;
				pCtrl->Step = 900;
			}
			break;

		case 900:	//Bw End
			pCtrl->ValveOut.ValveBw1 = 0;
			pCtrl->ValveOut.ValveBw2 = 0;

			pCtrl->p_set = 0;
			RClampCleanValveCtrl.p_set = 0;
			pCtrl->Step = 1000;
			break;

		case 1000:	//Inerval Timer Setting
			tValveClean->IN = 1;
			tValveClean->PT = pCleanValveFix->CleanValveInterval;
			pCtrl->Step = 1100;
			break;

		case 1100:	//Interval
			pCtrl->TimeDis.CleanValveIntervalDis = tValveClean->ET;
			if(1 == tValveClean->Q)
			{
				pCtrl->TimeDis.CleanValveIntervalDis = 0;
				tValveClean->IN = 0;
				pCtrl->Step = 1200;
			}
			break;

		case 1200:
			pCtrl->Step = 100;
			break;

		case 3000:
			tValveClean->IN      = 0;
			tValveCleanTotal->IN = 0;

			pCtrl->p_set = 0;
			pCtrl->ValveOut.ValveFw1 = 0;
			pCtrl->ValveOut.ValveFw2 = 0;

			pCtrl->ValveOut.ValveBw1 = 0;
			pCtrl->ValveOut.ValveBw2 = 0;

			pCtrl->Step = 0;
			break;
	}/* switch(pCtrl->Step) */

	pCtrl->TimeDis.CleanValveTotalDis = tValveCleanTotal->ET/60;

	if(1 == tValveCleanTotal->Q)
	{
		pCtrl->Step = 3000;
	}

}
```

#### clean.var
```iecst
VAR
	Step : UINT;
	keyOld : USINT;
	CleanValveTotalDis : UDINT;
	CleanValveFwDis : UDINT;
	CleanValveBwDis : UDINT;
	CleanValvePulse : BOOL;
	CleanValveIntervalDis : UDINT;
END_VAR
(*Clamp*)
VAR
	RClampCleanValveCtrl : CleanCtrl_typ;
	LClampCleanValveCtrl : CleanCtrl_typ;
END_VAR
(*Carriage*)
VAR
	RCarriageCleanValveCtrl : CleanCtrl_typ;
	LCarriageCleanValveCtrl : CleanCtrl_typ;
END_VAR
(*BlowPin*)
VAR
	RBlowPinCleanValveCtrl : CleanCtrl_typ;
	LBlowPinCleanValveCtrl : CleanCtrl_typ;
END_VAR
```

#### clean.typ - Local data types
```iecst
(********************************************************************
 * COPYRIGHT --
 ********************************************************************
 * Program: power
 * File: power.typ
 * Author: lij
 * Created: March 06, 2013
 ********************************************************************
 * Local data types of program power
 ********************************************************************)

TYPE
	CleanCtrl_typ : 	STRUCT
		Step : UINT;
		Enable : USINT;
		oldEnable : USINT;
		p_set : REAL;
		Para : CleanValvePara_typ;
		ValveOut : CleanValveOut_typ;
		TimeDis : CleanValveTimeDis_typ;
	END_STRUCT;
	CleanValveOut_typ : 	STRUCT
		ValveFw1 : USINT;
		ValveFw2 : USINT;
		ValveBw1 : USINT;
		ValveBw2 : USINT;
	END_STRUCT;
	CleanValveTimeDis_typ : 	STRUCT
		CleanValveTotalDis : UDINT;
		CleanValveFwDis : UDINT;
		CleanValveBwDis : UDINT;
		CleanValveIntervalDis : UDINT;
	END_STRUCT;
	CleanValvePara_typ : 	STRUCT
		P_FwClean : REAL;
		P_BwClean : REAL;
	END_STRUCT;
END_TYPE
```

- keyap880.h (reference to Logical/GlobalIncludes/keyap880.h)

### Package Logical/recipeMan - Recipe management

### recipeMan.var - Global variables
```iecst
(********************************************************************
 * COPYRIGHT --
 ********************************************************************
 * Package: recipeMag
 * File: recipeMag.var
 * Author: lij
 * Created: December 19, 2013
 ********************************************************************
 * Variables of package recipeMag
 ********************************************************************)
VAR CONSTANT
	C_MEM_MOLD_LENGTH : UINT := 12191;
	C_MEM_FIX_LENGTH : UINT := 12191;
	C_PVNAME_LENGTH : UINT := 31;
	C_LINE_NUMBER : UINT := 49;
END_VAR
```

### Program Logical/recipeMan/recipe (ANSIC, version 1.00.0) - recipe management

- recipe.h (reference to Logical/GlobalIncludes/recipe.h)

#### recipe.typ - Local data types
```iecst
(********************************************************************
 * COPYRIGHT --  B&R CHINA
 ********************************************************************
 * Program: recipe
 * File: recipe.typ
 * Author: lij
 * Created: March 06, 2013
 ********************************************************************
 * Local data types of program recipe
 ********************************************************************)

TYPE
	Text_Input_typ : 	STRUCT
		CurrentName : STRING[16];
		TempName : STRING[16];
		Text : STRING[2];
		SourceChar : STRING[80];
		Add : USINT;
		Del : USINT;
		Flash : USINT;
		Enable : USINT;
		Layer : USINT;
		Reserve : USINT;
	END_STRUCT;
	recipeButton_typ : 	STRUCT
		rename : USINT;
		save : USINT;
		open : USINT;
		clear : USINT;
		cancle : USINT;
		enter : USINT;
		Reserve2 : USINT;
		Reserve1 : USINT;
		former : USINT;
		next : USINT;
		lockFlag : UINT;
		lockListName : USINT;
	END_STRUCT;
	recipeName_typ : 	STRUCT
		recipeName : ARRAY[0..49]OF STRING[16];
		recipeTime : ARRAY[0..49]OF STRING[20];
		recipeIndex : UINT;
	END_STRUCT;
END_TYPE
```

#### recipe.var
```iecst
VAR
	DatObj_Info : DatObjInfo;
	DatObj_Create : DatObjCreate;
	DatObj_Write : DatObjWrite;
	DatObj_Read : DatObjRead;
	DataObjOperate : DatObj_Operate_typ;
	RecipeName : recipeName_typ;
	RecipeButton : recipeButton_typ;
	RecipeButtonNeg : recipeButton_typ;
	cntDealy : UDINT;
	RecordName : STRING[16];
	RecordTime : STRING[20];
	ListName : STRING[16];
	ListTime : STRING[20];
	ListIndex : USINT;
	RenameColor : UINT;
	ABCColor : ARRAY[0..79] OF UINT;
	KeyMatric : ARRAY[0..99] OF USINT;
	OldKeyMatric : ARRAY[0..99] OF USINT;
	OldLockFlag : USINT;
	i : UINT;
	iFlash : UINT;
	NumName : STRING[4];
	CurrentInput : INT;
	FiletypeUSB : USINT;
	StepRecipeUSB : UINT;
	cntTime : UINT;
	fileRecName : STRING[80];
	FileOpen_0 : FileOpen;
	FileCreate_0 : FileCreate;
	FileWrite_0 : FileWrite;
	FileRead_0 : FileRead;
	FileClose_0 : FileClose;
	bHideUSB_Key : USINT;
END_VAR
```

#### recipe.c
```c
/***********************************************************************************
 * COPYRIGHT -- B&R China
 ***********************************************************************************
 * Program: recipe
 * File: recipe.c
 * Author: lijianjun
 * Created: March 06, 2013
 ***********************************************************************************
 * Implementation of program recipe --- recipe management -load/save/clear
 **********************************************************************************/

#include <bur/plctypes.h>

#ifdef _DEFAULT_INCLUDES
	#include <AsDefault.h>
#endif

#include <string.h>

#include "edge.h"
#include "keyap2100.h"
//#include "keyap880.h"
#include "pic_id.h"
#include "recipe.h"

/***********************************************************************************
** 					 	         Macro Define								                **
***********************************************************************************/
#define S$STEP_INIT_OK     10000

#define S$STEP_IDLE        100
#define S$STEP_DM_READ     1000
#define S$STEP_DM_WRITE    2000
#define S$STEP_USB_READ    11000
#define S$STEP_USB_WRITE   12000
#define S$STEP_USB_CLOSE   13000

#define S$STEP_ERROR       30000

#define FILE_RECIPE_ALL         0
#define FILE_TYPE_ALL           1
#define FILE_TYPE_MOLD          2
#define FILE_TYPE_PROFILE       3
#define FILE_TYPE_MACHINE_FIX   4

/**********************************************************************************
**                            Function Declarations								      **
**********************************************************************************/
void InputMatric();

void KeyInputFun(unsigned short key,unsigned short current,Text_Input_typ * pInputCtrl);

/***********************************************************************************
**     	        		       I N I T U P  O F   T H E   T A S K 		 				 **
***********************************************************************************/
_INIT void receipe_init ( void )
{
	DataObjOperate.InitStep = 100;
	gRecipeOperate.NameOk   = 0;
	gRecipeOperate.DataOk   = 0;
	gRecipeOperate.CurveOk  = 0;

   strcpy(fileRecName, "nameAll.usb");		/* file name */

   strcpy(DataObjOperate.ModName,"recName");
	strcpy(DataObjOperate.Status,"Recipe name not start !");

   StepRecipeUSB = 0;
   cntTime = 0;

}/* end of _INIT */

/***********************************************************************************
**        				C Y C L I C   P A R T   O F   T H E   T A S K  			       **
***********************************************************************************/
 _CYCLIC void receipe_cyclic ( void )
{
   /* USB disk is insert or not  */
   gRecipeOperate.usbDiskOk = gUSB_1.DeviceOk | gUSB_2.DeviceOk;
   gRecipeOperate.bHideUSB  = !gRecipeOperate.usbDiskOk;

	/*  配方名字及数据初始化  */
	switch(DataObjOperate.InitStep)
	{
		case 100:
			/* Initialize info structure */
			DataObjOperate.Ident = 0;
			DatObj_Info.enable	= 1;
			DatObj_Info.pName	= (UDINT)DataObjOperate.ModName;

			/* Call  FUB  */
			DatObjInfo(&DatObj_Info);

			if(doERR_MODULNOTFOUND == DatObj_Info.status)
			{
				DataObjOperate.InitStep = 200;
			}
			else if(0 == DatObj_Info.status)
			{
				DataObjOperate.Ident = DatObj_Info.ident;
				DataObjOperate.InitStep  = 500;
			}
			else
			{
				DataObjOperate.InitStep = S$STEP_ERROR;
			}
			break;
		case 200:
			/* Initialize create structure */
			DatObj_Create.enable 	= 1;
			DatObj_Create.grp	 	   = 0;
			DatObj_Create.pName 	   = (UDINT)DataObjOperate.ModName;
			DatObj_Create.len 		= sizeof(RecipeName);
			DatObj_Create.MemType 	= doUSRROM;
			DatObj_Create.Option 	= 0;
			DatObj_Create.pCpyData 	= 0;

			/* Call FUB */
			DatObjCreate(&DatObj_Create);

			if(0 == DatObj_Create.status)
			{
				DataObjOperate.Ident = DatObj_Create.ident;
				DataObjOperate.InitStep = 300;
			}
			break;
		case 300:
			/*   Initialize Name structure info  */
			for (i=0;i<S$NUM_RECIPE;i++)
			{
            itoa((long)(i),(unsigned long)NumName);
				strcpy(RecipeName.recipeName[i],"recipe");
            strcat(RecipeName.recipeName[i],NumName);
				strcpy(RecipeName.recipeTime[i],"----.--.-- --:--");
			}
			DataObjOperate.InitStep = 400;
			break;
		case 400:
			/* Initialize write structure */
			DatObj_Write.enable  = 1;
			DatObj_Write.ident 	= DataObjOperate.Ident;
			DatObj_Write.Offset  = 0;
			DatObj_Write.pSource = (UDINT) &RecipeName;
			DatObj_Write.len 	 = sizeof (RecipeName);

			/* Call FUB */
			DatObjWrite(&DatObj_Write);

			if(0 == DatObj_Write.status)
			{
				DataObjOperate.InitStep = 500;
			}
			else
			{
				DataObjOperate.InitStep = S$STEP_ERROR;
			}
			break;
		case 500:
			/* Initialize read structure */
			DatObj_Read.enable = 1;
			DatObj_Read.ident  = DataObjOperate.Ident;
			DatObj_Read.Offset = 0;
			DatObj_Read.pDestination = (UDINT) &RecipeName;
			DatObj_Read.len = sizeof (RecipeName);

			/* Call FUB */
			DatObjRead(&DatObj_Read);

			if(0 == DatObj_Read.status)
			{
				DataObjOperate.InitStep = 600;
			}
			else
			{
				DataObjOperate.InitStep = S$STEP_ERROR;
			}
			break;
		case 600:		/*  load recipe name */
			if(strcmp(RecordName,"USB_FILE"))
			{
				gRecipeOperate.Index = RecipeName.recipeIndex;
				strcpy(RecordName,RecipeName.recipeName[gRecipeOperate.Index ]);
				strcpy(RecordTime,RecipeName.recipeTime[gRecipeOperate.Index ]);
			}
			else
			{
				gRecipeOperate.Index = S$NUM_RECIPE;
			}

			ListIndex = gRecipeOperate.Index ;
			strcpy(ListName,RecipeName.recipeName[ListIndex]);
			strcpy(ListTime,RecipeName.recipeTime[ListIndex]);
			DataObjOperate.InitStep = 700;
			break;
		case 700:       /*  load recipe data */
			gRecipeOperate.NameOk = 1;
			strcpy(DataObjOperate.Status,"Recipe name init ok !");
			DataObjOperate.Step     = S$STEP_IDLE;
			DataObjOperate.InitStep = S$STEP_INIT_OK;
			break;
		case S$STEP_INIT_OK:
			break;

		case S$STEP_ERROR:
			break;

		default:
			break;
	}/* switch(DataObjOperate.InitStep) */

	if((0 == DataObjOperate.Ident)||( gPanelObj.GetPicture != PIC_RECIPE)||
	   (DataObjOperate.InitStep != S$STEP_INIT_OK ))
	{
		cntDealy = 10;

		RecipeButton.lockFlag     = 0;
		RecipeButton.lockListName = 0;
		RecipeButton.rename   	  = 0;
		RecipeButton.save         = 0;
		RecipeButton.open         = 0;
		RecipeButton.clear        = 0;
		RecipeButton.former       = 0;
		RecipeButton.next         = 0;
		RecipeButtonNeg = RecipeButton;

      gPanelObj.SetKeyLevel = 0;
		return;
	}
	else
	{
		if(cntDealy > 0)
		{
			cntDealy--;
			return;
		}

		if(EDGEPOS(gPanelObj.KeyMatric[S$KEYMATRIX_F11],OldKeyMatric[S$KEYMATRIX_F11]) && gPanelObj.PasswordLevel >0)
		{
			gImply.InfoRecipe = 1;
			RecipeButton.rename = 1;
		}
		if(EDGEPOS(gPanelObj.KeyMatric[S$KEYMATRIX_F12],OldKeyMatric[S$KEYMATRIX_F12])&& gPanelObj.PasswordLevel >0)
		{
			gImply.InfoRecipe = 1;
			RecipeButton.save = 1;
		}
		if(EDGEPOS(gPanelObj.KeyMatric[S$KEYMATRIX_F13],OldKeyMatric[S$KEYMATRIX_F13]))
		{
			gImply.InfoRecipe = 1;
			RecipeButton.open = 1;
		}
		if(EDGEPOS(gPanelObj.KeyMatric[S$KEYMATRIX_F14],OldKeyMatric[S$KEYMATRIX_F14])&& gPanelObj.PasswordLevel >0)
		{
			gImply.InfoRecipe = 1;
			RecipeButton.clear = 1;
		}

		RecipeButton.cancle = gPanelObj.KeyMatric[S$KEYMATRIX_ESC];
		RecipeButton.enter  = gPanelObj.KeyMatric[S$KEYMATRIX_ENTER];

      /* recipe in USB disk file button  */
      if(1 == gRecipeOperate.usbDiskOk)
      {
			if(1 == gRecipeOperate.NameLoad)
			{
				gRecipeOperate.NameLoad = 0;
				strcpy(RecordName,"USB_FILE");
				strcpy(RecordTime,gPanelObj.CurrentTime);
				gRecipeOperate.Index = S$NUM_RECIPE;
			}
			if (gPanelObj.PasswordLevel<4) //ipis0226
			{
				FiletypeUSB=FILE_TYPE_ALL;
			}
         bHideUSB_Key = 0;
         switch(FiletypeUSB)
         {
            case FILE_TYPE_ALL:
               if((gUSB_1.DeviceOk == 1) || (gUSB_2.DeviceOk == 1))
               {
                  if(gUSB_1.DeviceOk == 1)
                  {
                     strcpy(gRecipeOperate.deviceNameUSB, gUSB_1.DirSingleDeviceName);
                  }
                  else if(gUSB_2.DeviceOk == 1)
                  {
                     strcpy(gRecipeOperate.deviceNameUSB, gUSB_2.DirSingleDeviceName);
                  }
               }/* if((gUSB_1.DeviceOk == 1) || (gUSB_2.DeviceOk == 1)) */

               if(StepRecipeUSB != 0)bHideUSB_Key = 1;

               if(EDGEPOS(gPanelObj.KeyMatric[S$KEYMATRIX_F4],OldKeyMatric[S$KEYMATRIX_F4]))
               {
                 // if(0 == StepRecipeUSB)StepRecipeUSB = 100;
					if(0 == StepRecipeUSB)StepRecipeUSB = 120;  //ipis0226
               }
               if(EDGEPOS(gPanelObj.KeyMatric[S$KEYMATRIX_F5],OldKeyMatric[S$KEYMATRIX_F5]))
               {
                //  if(0 == StepRecipeUSB)StepRecipeUSB = 200;
				if(0 == StepRecipeUSB)StepRecipeUSB = 220;	  //ipis0226
               }
               break;

            case FILE_TYPE_MOLD:
               if((gUSB_1.DeviceOk == 1) || (gUSB_2.DeviceOk == 1))
               {
                  if(gUSB_1.DeviceOk == 1)
                  {
                     strcpy(gRecipeOperate.deviceNameUSB, gUSB_1.DirSingleDeviceName);
                  }
                  else if(gUSB_2.DeviceOk == 1)
                  {
                     strcpy(gRecipeOperate.deviceNameUSB, gUSB_2.DirSingleDeviceName);
                  }
               }/* if((gUSB_1.DeviceOk == 1) || (gUSB_2.DeviceOk == 1)) */

               bHideUSB_Key = !gRecipeOperate.usbMoldOk;

               if(EDGEPOS(gPanelObj.KeyMatric[S$KEYMATRIX_F4],OldKeyMatric[S$KEYMATRIX_F4]))
               {
                  if(1 == gRecipeOperate.usbMoldOk)gRecipeOperate.DataUSBSave = 1;
               }
               if(EDGEPOS(gPanelObj.KeyMatric[S$KEYMATRIX_F5],OldKeyMatric[S$KEYMATRIX_F5]))
               {
                  if(1 == gRecipeOperate.usbMoldOk)gRecipeOperate.DataUSBLoad = 1;
               }
               break;

            case FILE_TYPE_PROFILE:
               if((gUSB_1.DeviceOk == 1) || (gUSB_2.DeviceOk == 1))
               {
                  if(gUSB_1.DeviceOk == 1)
                  {
                     strcpy(gRecipeOperate.deviceNameUSB, gUSB_1.DirSingleDeviceName);
                  }
                  else if(gUSB_2.DeviceOk == 1)
                  {
                     strcpy(gRecipeOperate.deviceNameUSB, gUSB_2.DirSingleDeviceName);
                  }
               }/* if((gUSB_1.DeviceOk == 1) || (gUSB_2.DeviceOk == 1)) */

               bHideUSB_Key = !gRecipeOperate.usbCurveOk;

               if(EDGEPOS(gPanelObj.KeyMatric[S$KEYMATRIX_F4],OldKeyMatric[S$KEYMATRIX_F4]))
               {
                  if(1 == gRecipeOperate.usbCurveOk)gRecipeOperate.CurveUSBSave = 1;
               }
               if(EDGEPOS(gPanelObj.KeyMatric[S$KEYMATRIX_F5],OldKeyMatric[S$KEYMATRIX_F5]))
               {
                  if(1 == gRecipeOperate.usbCurveOk)gRecipeOperate.CurveUSBLoad = 1;
               }
               break;

            case FILE_TYPE_MACHINE_FIX:
               if((gUSB_1.DeviceOk == 1) || (gUSB_2.DeviceOk == 1))
               {
                  if(gUSB_1.DeviceOk == 1)
                  {
                     strcpy(gRecipeOperate.deviceNameUSB, gUSB_1.DirSingleDeviceName);
                  }
                  else if(gUSB_2.DeviceOk == 1)
                  {
                     strcpy(gRecipeOperate.deviceNameUSB, gUSB_2.DirSingleDeviceName);
                  }
               }/* if((gUSB_1.DeviceOk == 1) || (gUSB_2.DeviceOk == 1)) */

               bHideUSB_Key = !gRecipeOperate.usbFixOk;

               if(EDGEPOS(gPanelObj.KeyMatric[S$KEYMATRIX_F4],OldKeyMatric[S$KEYMATRIX_F4]))
               {
                  if(1 == gRecipeOperate.usbFixOk)gRecipeOperate.OnceUSBSave = 1;
               }
               if(EDGEPOS(gPanelObj.KeyMatric[S$KEYMATRIX_F5],OldKeyMatric[S$KEYMATRIX_F5]))
               {
                  if(1 == gRecipeOperate.usbFixOk)gRecipeOperate.OnceUSBLoad = 1;
               }
               break;

            case FILE_RECIPE_ALL:
               if((gUSB_1.DeviceOk == 1) || (gUSB_2.DeviceOk == 1))
               {
                  if(gUSB_1.DeviceOk == 1)
                  {
                     strcpy(gRecipeOperate.deviceNameUSB, gUSB_1.DirAllDeviceName);
                  }
                  else if(gUSB_2.DeviceOk == 1)
                  {
                     strcpy(gRecipeOperate.deviceNameUSB, gUSB_2.DirAllDeviceName);
                  }
               }/* if((gUSB_1.DeviceOk == 1) || (gUSB_2.DeviceOk == 1)) */

               if(StepRecipeUSB != 0)bHideUSB_Key = 1;

               if(EDGEPOS(gPanelObj.KeyMatric[S$KEYMATRIX_F4],OldKeyMatric[S$KEYMATRIX_F4]))
               {
                  if(0 == StepRecipeUSB)StepRecipeUSB = 1100;
               }
               if(EDGEPOS(gPanelObj.KeyMatric[S$KEYMATRIX_F5],OldKeyMatric[S$KEYMATRIX_F5]))
                  {
                  if(0 == StepRecipeUSB)StepRecipeUSB = 1200;
               }
               break;
         }/* switch(FiletypeUSB) */

         /* step machine to save / load USB pecipe  */
         switch(StepRecipeUSB)
         {
            case 0:
               cntTime = 0;
               break;

            /* save current recipe to USB disk */
            case 100:
               gRecipeOperate.OnceUSBSave = 1;
               cntTime = 0;
               StepRecipeUSB = 110;
               break;

            case 110:
               cntTime = cntTime + 1;
               if(cntTime > 10 && 1 == gRecipeOperate.usbFixOk)
               {
                  cntTime = 0;
                  StepRecipeUSB = 120;
               }
               break;

            case 120:
               gRecipeOperate.DataUSBSave = 1;
               cntTime = 0;
               StepRecipeUSB = 130;
               break;

            case 130:
               cntTime = cntTime + 1;
               if(cntTime > 10 && 1 == gRecipeOperate.usbMoldOk)
               {
                  cntTime = 0;
                  StepRecipeUSB = 140;
               }
               break;

            case 140:
               gRecipeOperate.CurveUSBSave = 1;
               cntTime = 0;
               StepRecipeUSB = 150;
               break;

            case 150:
               cntTime = cntTime + 1;
               if(cntTime > 30 && 1 == gRecipeOperate.usbCurveOk)
               {
                  cntTime = 0;
                  StepRecipeUSB = 0;
               }
               break;

            /* load current recipe from USB disk */
            case 200:
               gRecipeOperate.OnceUSBLoad = 1;
               cntTime = 0;
               StepRecipeUSB = 210;
               break;

            case 210:
               cntTime = cntTime + 1;
               if(cntTime > 10 && 1 == gRecipeOperate.usbFixOk)
               {
                  cntTime = 0;
                  StepRecipeUSB = 220;
               }
               break;

            case 220:
               gRecipeOperate.DataUSBLoad = 1;
               cntTime = 0;
               StepRecipeUSB = 230;
               break;

            case 230:
               cntTime = cntTime + 1;
               if(cntTime > 10 && 1 == gRecipeOperate.usbMoldOk)
               {
                  cntTime = 0;
                  StepRecipeUSB = 240;
               }
               break;

            case 240:
               gRecipeOperate.CurveUSBLoad = 1;
               cntTime = 0;
               StepRecipeUSB = 250;
               break;

            case 250:
               cntTime = cntTime + 1;
               if(cntTime > 30 && 1 == gRecipeOperate.usbCurveOk)
               {
                  cntTime = 0;
                  StepRecipeUSB = 0;
               }
               break;

            /* ------------------------------- */
            /*   save all recipe to USB disk   */
            /* ------------------------------- */
            case 1100:
               gRecipeOperate.OnceUSBSave = 1;
               cntTime = 0;
               StepRecipeUSB = 1110;
               break;

            case 1110:
               cntTime = cntTime + 1;
               if(cntTime > 10 && 1 == gRecipeOperate.usbFixOk)
               {
                  cntTime = 0;
                  StepRecipeUSB = 1120;
               }
               break;

            case 1120:
               gRecipeOperate.DataUSBSaveAll = 1;
               cntTime = 0;
               StepRecipeUSB = 1130;
               break;

            case 1130:
               cntTime = cntTime + 1;
               if(cntTime > 10 && 1 == gRecipeOperate.usbMoldOk)
               {
                  cntTime = 0;
                  StepRecipeUSB = 1140;
               }
               break;

            case 1140:
               gRecipeOperate.CurveUSBSaveAll = 1;
               cntTime = 0;
               StepRecipeUSB = 1150;
               break;

            case 1150:
               cntTime = cntTime + 1;
               if(cntTime > 30 && 1 == gRecipeOperate.usbCurveOk)
               {
                  cntTime = 0;
                  StepRecipeUSB = 1160;
               }
               break;

            case 1160:
               DataObjOperate.Step = S$STEP_USB_WRITE;
               cntTime = 0;
               StepRecipeUSB = 1170;
               break;

            case 1170:
               cntTime = cntTime + 1;
               if(cntTime > 20 && S$STEP_IDLE == DataObjOperate.Step)
               {
                  cntTime = 0;
                  StepRecipeUSB = 0;
               }
               break;

            /* --------------------------------- */
            /*    load all recipe from USB disk  */
            /* --------------------------------- */
            case 1200:
               gRecipeOperate.OnceUSBLoad = 1;
               cntTime = 0;
               StepRecipeUSB = 1210;
               break;

            case 1210:
               cntTime = cntTime + 1;
               if(cntTime > 10 && 1 == gRecipeOperate.usbFixOk)
               {
                  cntTime = 0;
                  StepRecipeUSB = 1220;
               }
               break;

            case 1220:
               gRecipeOperate.DataUSBLoadAll = 1;
               cntTime = 0;
               StepRecipeUSB = 1230;
               break;

            case 1230:
               cntTime = cntTime + 1;
               if(cntTime > 10 && 1 == gRecipeOperate.usbMoldOk)
               {
                  cntTime = 0;
                  StepRecipeUSB = 1240;
               }
               break;

            case 1240:
               gRecipeOperate.CurveUSBLoadAll = 1;
               cntTime = 0;
               StepRecipeUSB = 1250;
               break;

            case 1250:
               cntTime = cntTime + 1;
               if(cntTime > 30 && 1 == gRecipeOperate.usbCurveOk)
               {
                  cntTime = 0;
                  StepRecipeUSB = 1260;
               }
               break;

            case 1260:
               DataObjOperate.Step = S$STEP_USB_READ;
               cntTime = 0;
               StepRecipeUSB = 1270;
               break;

            case 1270:
               cntTime = cntTime + 1;
               if(cntTime > 20 && S$STEP_IDLE == DataObjOperate.Step)
               {
                  cntTime = 0;
                  StepRecipeUSB = 0;
               }
               break;
         }/* switch(StepRecipeUSB) */

      }/* if(1 == gImply.usbDiskOk) */
      else
      {
         bHideUSB_Key = 1;
         cntTime = 0;
         StepRecipeUSB = 0;
      }
	} /* if((0 == DataObjOperate.Ident)||( gPanelObj.GetPicture != PIC_RECIPE)||
	   (DataObjOperate.InitStep != S$STEP_INIT_OK )) */

	if(1 == RecipeButton.lockFlag)
	{
      gPanelObj.SetKeyLevel = 0;
		RenameColor = 0x0016;  /* 黄底黑字 */
	}
	else
	{
      gPanelObj.SetKeyLevel = 0;
		RenameColor = 0x0007;  	/* 灰底黑字 */

      for(i=0;i<10;i++)
      {
         ABCColor[i]    = 0x0707;
         ABCColor[10+i] = 0x0707;
         ABCColor[20+i] = 0x0707;
         ABCColor[30+i] = 0x0707;
         ABCColor[40+i] = 0x0707;
         ABCColor[50+i] = 0x0707;
         ABCColor[60+i] = 0x0707;
      }

		strcpy(ListName,RecipeName.recipeName[ListIndex]);

		if(0 == RecipeButton.lockFlag)
		{
			RecipeButton.former = gPanelObj.KeyMatric[S$KEYMATRIX_UP];
			RecipeButton.next   = gPanelObj.KeyMatric[S$KEYMATRIX_DOWN];
		}
		else
		{
			RecipeButton.former = 0;
			RecipeButton.next   = 0;
		}
	}

	OldLockFlag = RecipeButton.lockFlag;

	switch(DataObjOperate.Step)
	{
		case S$STEP_IDLE:
			if(0 == RecipeButton.lockFlag)
			{
				if (EDGENEG(RecipeButton.former,RecipeButtonNeg.former))
				{
					if (ListIndex > 0)
					{
						ListIndex--;
					}
					else
					{
						ListIndex = S$NUM_RECIPE - 1;
					}

					strcpy(ListName,RecipeName.recipeName[ListIndex]);
					strcpy(ListTime,RecipeName.recipeTime[ListIndex]);
				}
				if (EDGENEG(RecipeButton.next,RecipeButtonNeg.next))
				{
					if (ListIndex < (S$NUM_RECIPE - 1))
					{
						ListIndex++;
					}
					else
					{
						ListIndex = 0;
					}

					strcpy(ListName,RecipeName.recipeName[ListIndex]);
					strcpy(ListTime,RecipeName.recipeTime[ListIndex]);
				}

				if (1 == RecipeButton.rename)
				{
					RecipeButton.lockFlag = 1;
				}

				if (1 == RecipeButton.save)
				{
					RecipeButton.lockFlag = 2;
				}

				if (1 == RecipeButton.open)
				{
					RecipeButton.lockFlag = 3;
				}

				if (1 == RecipeButton.clear)
				{
					RecipeButton.lockFlag = 4;
				}

				if(1 == RecipeButton.rename)
				{
					RecipeButton.lockListName = 1;
				}
				else
				{
					RecipeButton.lockListName = 0;
				}
			}/* if(0 == RecipeButton.lockFlag) */
			else if(1 == RecipeButton.lockFlag)
			{
				RecipeButton.save   = 0;
				RecipeButton.open   = 0;
				RecipeButton.clear  = 0;
			}
			else if(2 == RecipeButton.lockFlag)
			{
				RecipeButton.rename = 0;
				RecipeButton.open   = 0;
				RecipeButton.clear  = 0;
			}
			else if(3 == RecipeButton.lockFlag)
			{
				RecipeButton.rename = 0;
				RecipeButton.save   = 0;
				RecipeButton.clear  = 0;
			}
			else
			{
				RecipeButton.rename = 0;
				RecipeButton.save   = 0;
				RecipeButton.open  = 0;
			}

			/*  Assert operation   */
			if (EDGENEG(RecipeButton.enter,RecipeButtonNeg.enter))
			{
				switch(RecipeButton.lockFlag)
				{
					case 1:              /*  rename  */
						strcpy(RecipeName.recipeName[ListIndex],ListName/*TextInput.CurrentName*/);
						if(ListIndex == gRecipeOperate.Index)strcpy(RecordName,ListName/*TextInput.CurrentName*/);
						DataObjOperate.Step = S$STEP_DM_WRITE;
						break;
					case 2:              /*  save  */
						/*  set recipe data from current*/
						gRecipeOperate.Index = ListIndex;
				RecipeName.recipeIndex = gRecipeOperate.Index;
						strcpy(RecordTime,gPanelObj.CurrentTime);
                  strcpy(RecordName,RecipeName.recipeName[gRecipeOperate.Index]);
						strcpy(RecipeName.recipeTime[gRecipeOperate.Index],gPanelObj.CurrentTime);
                  gRecipeOperate.CurveRecipeSave = 1;
                  gRecipeOperate.DataRecipeSave  = 1;
                  gRecipeOperate.OnceSave = 1;
                  DataObjOperate.Step = S$STEP_DM_WRITE;
						break;
					case 3:              /*  open  */
						gRecipeOperate.Index = ListIndex;
						RecipeName.recipeIndex = gRecipeOperate.Index;

						strcpy(RecordName,RecipeName.recipeName[gRecipeOperate.Index]);
						strcpy(RecordTime,RecipeName.recipeTime[gRecipeOperate.Index]);

						strcpy(ListName,RecipeName.recipeName[ListIndex]);
						strcpy(ListTime,RecipeName.recipeTime[ListIndex]);
						/*  load recipe data */
                  gRecipeOperate.CurveRecipeLoad = 1;
                  gRecipeOperate.DataRecipeLoad  = 1;
                  gRecipeOperate.OnceLoad = 1;
                  DataObjOperate.Step = S$STEP_DM_READ;
						break;
					case 4:              /*  clear  */
						if(gRecipeOperate.Index != ListIndex)
						{
							strcpy(RecipeName.recipeName[ListIndex],"Recipe");
							strcpy(RecipeName.recipeTime[ListIndex],"----.--.-- --:--");
							DataObjOperate.Step = S$STEP_DM_WRITE;
							/*  set recipe data  0*/
						}
						break;
				}/* switch(RecipeButton.lockFlag) */

				RecipeButton.lockFlag = 0;
				RecipeButton.rename   = 0;
				RecipeButton.save     = 0;
				RecipeButton.open     = 0;
				RecipeButton.clear    = 0;
			}/* (EDGENEG(RecipeButton.enter,RecipeButtonNeg.enter)) */

			/*cancle any operation */
			if(EDGENEG(RecipeButton.cancle,RecipeButtonNeg.cancle))
			{
				if(1 == RecipeButton.lockFlag)
				{
					strcpy(ListName,RecipeName.recipeName[ListIndex]);
					strcpy(ListTime,RecipeName.recipeTime[ListIndex]);
				}
				RecipeButton.lockFlag = 0;
				RecipeButton.rename   = 0;
				RecipeButton.save     = 0;
				RecipeButton.open     = 0;
				RecipeButton.clear    = 0;
			}

			if(1 == gRecipeOperate.NameSave)
			{
				gRecipeOperate.NameSave = 0;
				DataObjOperate.Step = S$STEP_DM_WRITE;
			}
			break; /* S$STEP_IDLE:  */

		case S$STEP_DM_READ:
			DataObjOperate.Step = S$STEP_DM_READ + 100;
			strcpy(DataObjOperate.Status,"Recipe name read ok !");
			break;

		case (S$STEP_DM_READ + 100):
			DataObjOperate.Step = S$STEP_IDLE;
			break;

		case S$STEP_DM_WRITE:
			strcpy(DataObjOperate.Status,"");
			DatObj_Write.enable = 1;
			DatObj_Write.ident 	= DataObjOperate.Ident;
			DatObj_Write.Offset = 0;
			DatObj_Write.pSource = (UDINT) &RecipeName;
			DatObj_Write.len 	 = sizeof (RecipeName);

			/* Call FUB */
			DatObjWrite(&DatObj_Write);

			if(0 == DatObj_Write.status)
			{
				DataObjOperate.Step = S$STEP_DM_WRITE + 100;
			}
			else
			{
				DataObjOperate.Step = S$STEP_IDLE;
			}
			break;

		case (S$STEP_DM_WRITE + 100):
			DataObjOperate.Step = S$STEP_IDLE;
			if(0 == DatObj_Write.status)
			{
				strcpy(DataObjOperate.Status,"Recipe name write ok !");
			}
			else
			{
				strcpy(DataObjOperate.Status,"Recipe name write false !");
			}
			break;

      /* ------------------------------------------------- */
      /* ----------------- save to USB disk -------------- */
      /* ------------------------------------------------- */
      case S$STEP_USB_WRITE:
         FileOpen_0.enable  = 1;
         FileOpen_0.pDevice = (UDINT)&gRecipeOperate.deviceNameUSB;
         FileOpen_0.pFile   = (UDINT)&fileRecName;
         FileOpen_0.mode    = fiREAD_WRITE;

         /* Call FUB */
         FileOpen(&FileOpen_0);

         if(fiERR_FILE_NOT_FOUND == FileOpen_0.status)/* no file   */
         {
            FileOpen_0.enable  = 0;
            DataObjOperate.Step = S$STEP_USB_WRITE + 100;
         }
         else
         {
            if(ERR_OK == FileOpen_0.status)			/* file exist */
            {
               FileOpen_0.enable  = 0;
               if(FileOpen_0.filelen == sizeof(RecipeName))
               {
                  DataObjOperate.IdentUSB = FileOpen_0.ident;
                  DataObjOperate.Step = S$STEP_USB_WRITE + 200;
               }
               else
               {
                  DataObjOperate.Step = S$STEP_USB_CLOSE;
               }
            }
            else if (FileOpen_0.status != ERR_FUB_BUSY)
            {
               FileOpen_0.enable  = 0;
               DataObjOperate.Step = S$STEP_ERROR;
            }
         }
         break;

      case (S$STEP_USB_WRITE + 100):
         FileCreate_0.enable  = 1;
         FileCreate_0.pDevice = (UDINT)&gRecipeOperate.deviceNameUSB;
         FileCreate_0.pFile   = (UDINT)&fileRecName;

         /* Call FUB */
         FileCreate(&FileCreate_0);

         if(ERR_OK == FileCreate_0.status)		/* ok */
         {
            FileCreate_0.enable = 0;
            DataObjOperate.IdentUSB = FileCreate_0.ident;
            DataObjOperate.Step = S$STEP_USB_WRITE + 200;
         }
         else if (FileCreate_0.status != ERR_FUB_BUSY)
         {
            FileCreate_0.enable= 0;
            DataObjOperate.Step = S$STEP_USB_CLOSE;
         }
        break;

      case (S$STEP_USB_WRITE + 200):
         FileWrite_0.enable = 1;
         FileWrite_0.ident  = DataObjOperate.IdentUSB;
         FileWrite_0.offset = 0;
         FileWrite_0.pSrc   = (UDINT)&RecipeName;
         FileWrite_0.len    = sizeof(RecipeName);

         /* Call FUB */
         FileWrite(&FileWrite_0);

         if(ERR_OK == FileWrite_0.status)				/* ok */
         {
            FileWrite_0.enable = 0;
            DataObjOperate.Step = S$STEP_USB_CLOSE;
         }
         else if (FileWrite_0.status != ERR_FUB_BUSY)
         {
            FileWrite_0.enable = 0;
            DataObjOperate.Step = S$STEP_USB_CLOSE;
         }
         break;

      /* ------------------------------------------------- */
      /* ----------------- Load from USB disk ------------ */
      /* ------------------------------------------------- */
      case S$STEP_USB_READ:
         FileOpen_0.enable  = 1;
         FileOpen_0.pDevice = (UDINT)&gRecipeOperate.deviceNameUSB;
         FileOpen_0.pFile   = (UDINT)&fileRecName;
         FileOpen_0.mode    = fiREAD_WRITE;

         /* Call FUB */
         FileOpen(&FileOpen_0);

         if(fiERR_FILE_NOT_FOUND == FileOpen_0.status)	/* no file   */
         {
            FileOpen_0.enable  = 0;
            DataObjOperate.Step = S$STEP_IDLE;
         }
         else
         {
            if(ERR_OK == FileOpen_0.status)				/* file exist */
            {
               FileOpen_0.enable = 0;
               if(FileOpen_0.filelen == sizeof(RecipeName))
               {
                  DataObjOperate.IdentUSB = FileOpen_0.ident;
                  DataObjOperate.Step = S$STEP_USB_READ + 100;
               }
               else
               {
                  DataObjOperate.Step = S$STEP_USB_CLOSE;
               }
            }
            else if (FileOpen_0.status != ERR_FUB_BUSY)
            {
               FileOpen_0.enable = 0;
               DataObjOperate.Step = S$STEP_ERROR;
            }
         }
         break;

      case (S$STEP_USB_READ + 100):
         FileRead_0.enable = 1;
         FileRead_0.ident  = DataObjOperate.IdentUSB;
         FileRead_0.offset = 0;
         FileRead_0.pDest  = (UDINT)&RecipeName;
         FileRead_0.len    = sizeof(RecipeName);

         /* Call FUB */
         FileRead(&FileRead_0);

         if(ERR_OK == FileRead_0.status)	/* ok */
         {
            FileRead_0.enable = 0;
				gRecipeOperate.NameSave = 1;
            DataObjOperate.Step = S$STEP_USB_CLOSE;
         }
         else
         {
            FileRead_0.enable = 0;
            DataObjOperate.Step = S$STEP_USB_CLOSE;
         }
         break;
      /* ------------------------------------------------------- */
      /* ---------------- Close USB file device ---------------- */
      /* ------------------------------------------------------- */
      case S$STEP_USB_CLOSE:
         FileClose_0.enable = 1;
         FileClose_0.ident  = DataObjOperate.IdentUSB;

         /* Call FBK */
         FileClose(&FileClose_0);

         if(ERR_OK == FileClose_0.status)	/* ok */
         {
            FileClose_0.enable = 0;
            DataObjOperate.Step =  S$STEP_IDLE;
         }
         else if (FileClose_0.status != ERR_FUB_BUSY)
         {
            FileClose_0.enable = 0;
            DataObjOperate.Step = S$STEP_ERROR;
         }
         break;

		case S$STEP_ERROR:
			DataObjOperate.Step = S$STEP_IDLE;
			break;
	}/* switch(DataObjOperate.Step) */

	if(0 == RecipeButton.rename && 0 == RecipeButton.save &&
	   0 == RecipeButton.open   && 0 == RecipeButton.clear)
	{
		RecipeButton.lockFlag = 0;
	}
	RecipeButtonNeg = RecipeButton;
}
/**************************************************************************************/
void InputMatric()
{
	if(1 == gPanelObj.KeyMatric[S$KEYMATRIX_NUM0])
	{
		CurrentInput ++ ;
		if(CurrentInput < 63)
		{
			CurrentInput = 63;
		}

		if(CurrentInput > 69)
		{
			CurrentInput = 63;
		}

	}

	if(1 == gPanelObj.KeyMatric[S$KEYMATRIX_NUM1])
	{
		CurrentInput ++ ;
		if(CurrentInput < 0)
		{
			CurrentInput = 0;
		}

		if(CurrentInput > 6)
		{
			CurrentInput = 0;
		}
	}

	if(1 ==gPanelObj.KeyMatric[S$KEYMATRIX_NUM2])
	{
		CurrentInput ++ ;
		if(CurrentInput < 7)
		{
			CurrentInput = 7;
		}

		if(CurrentInput > 13)
		{
			CurrentInput = 7;
		}
	}

	if(1 == gPanelObj.KeyMatric[S$KEYMATRIX_NUM3])
	{
		CurrentInput ++ ;
		if(CurrentInput < 14)
		{
			CurrentInput = 14;
		}

		if(CurrentInput > 20)
		{
			CurrentInput = 14;
		}
	}
	if(1 == gPanelObj.KeyMatric[S$KEYMATRIX_NUM4])
	{
		CurrentInput ++ ;
		if(CurrentInput < 21)
		{
			CurrentInput = 21;
		}

		if(CurrentInput > 27)
		{
			CurrentInput = 21;
		}
	}

	if(1 == gPanelObj.KeyMatric[S$KEYMATRIX_NUM5])
	{
		CurrentInput ++ ;
		if(CurrentInput < 28)
		{
			CurrentInput = 28;
		}

		if(CurrentInput > 34)
		{
			CurrentInput = 28;
		}
	}

	if(1 == gPanelObj.KeyMatric[S$KEYMATRIX_NUM6])
	{
		CurrentInput ++ ;
		if(CurrentInput < 35)
		{
			CurrentInput = 35;
		}

		if(CurrentInput > 41)
		{
			CurrentInput = 35;
		}
	}

	if(1 == gPanelObj.KeyMatric[S$KEYMATRIX_NUM7])
	{
		CurrentInput ++ ;
		if(CurrentInput < 42)
		{
			CurrentInput = 42;
		}

		if(CurrentInput > 48)
		{
			CurrentInput = 42;
		}
	}

	if(1 == gPanelObj.KeyMatric[S$KEYMATRIX_NUM8])
	{
		CurrentInput ++ ;
		if(CurrentInput < 49)
		{
			CurrentInput = 49;
		}

		if(CurrentInput > 55)
		{
			CurrentInput = 49;
		}
	}

	if(1 == gPanelObj.KeyMatric[S$KEYMATRIX_NUM9])
	{
		CurrentInput ++ ;
		if(CurrentInput < 56)
		{
			CurrentInput = 56;
		}

		if(CurrentInput > 62)
		{
			CurrentInput = 56;
		}
	}

	if(1 == gPanelObj.KeyMatric[S$KEYMATRIX_DOWN])
	{
		CurrentInput = CurrentInput + 7;
		if(CurrentInput > 70)CurrentInput = CurrentInput - 70;
	}

	if(1 == gPanelObj.KeyMatric[S$KEYMATRIX_UP])
	{
		CurrentInput = CurrentInput - 7;
		if(CurrentInput < 0)CurrentInput = CurrentInput + 70;
	}

	if(1 == gPanelObj.KeyMatric[S$KEYMATRIX_LEFT])
	{
		CurrentInput = CurrentInput - 1;
		if((CurrentInput % 7) == 0)CurrentInput = CurrentInput + 7;
	}

	if(1 == gPanelObj.KeyMatric[S$KEYMATRIX_RIGHT])
	{
		CurrentInput = CurrentInput + 1;
		if((CurrentInput % 7) == 0)CurrentInput = CurrentInput - 7;
	}

	if(CurrentInput < 0)CurrentInput= 0;
	if(CurrentInput > 69)CurrentInput =69;
}
void KeyInputFun(unsigned short key,unsigned short current, Text_Input_typ * pInputCtrl)
{

	strcpy(pInputCtrl->SourceChar,"1ABCabc2DEFdef3GHIghi4JKLjhl5MNOmno6PQRpqr7STUstu8VWXvwz9YZyz-.0*/()[]        ");

	if(1 == EDGEPOS(gPanelObj.KeyMatric[key],KeyMatric[key]))
	{
		switch (key)
		{
			case S$KEYMATRIX_TAB:
				if(strlen(pInputCtrl->CurrentName) < 12)
				{
					strcpy(pInputCtrl->Text,"");
					memcpy(pInputCtrl->Text,pInputCtrl->SourceChar+current,1);
					strcat(pInputCtrl->CurrentName,pInputCtrl->Text);
				}
				break;
			case S$KEYMATRIX_DEL:
				if(strlen(pInputCtrl->CurrentName) > 0)
				{
					memset(pInputCtrl->CurrentName + strlen(pInputCtrl->CurrentName)- 1,0,1);
				}
				break;
			case S$KEYMATRIX_ENTER:
				pInputCtrl->Flash = 0;
				break;
			default:
				break;
		}

	}

	if (1 == pInputCtrl->Flash)
    {
 		iFlash++;
 		if(iFlash > 6)iFlash=0;

	 	if (iFlash  < 3)
	 	{
	    	strcpy(pInputCtrl->TempName,pInputCtrl->CurrentName);
	 		strcat(pInputCtrl->TempName, "_");
	 	}
	 	else
	 	{
	    	strcpy(pInputCtrl->TempName,pInputCtrl->CurrentName);
	 		strcat(pInputCtrl->TempName, " ");
	 	}
 	}
 	else
 	{
 		strcpy(pInputCtrl->TempName,pInputCtrl->CurrentName);
 	}

	for(i = strlen(pInputCtrl->TempName);i<14;i++)
	{
		pInputCtrl->TempName[i] = ' ';
	}
}
```

### Program Logical/recipeMan/multsave (ANSIC, version 1.00.0) - mold data load/save
